// TIA Portal V19 export
DATA_BLOCK "A0201_Profilatrice_RegolazioneFormato_PERS"   // DB70
// stored: MemoryReserve 100
   VAR RETAIN
      Par_Machine { ExternalAccessible := 'False'; ExternalVisible := 'False'; ExternalWritable := 'False'} : Struct
         Passaggio02_MaxDisallineamentoAXs : Real := 0.5;   // (Controllo disabilitato se <= 0)
         Passaggio14_MaxDisallineamentoAXs : Real := 0.5;   // (Controllo disabilitato se <= 0)
         Passaggio17_MaxDisallineamentoAXs : Real := 0.5;   // (Controllo disabilitato se <= 0)
         Passaggio18_MaxDisallineamentoAXs : Real := 0.5;   // (Controllo disabilitato se <= 0)
         AxD_AutoSpeed : Real := 100.0;
      END_STRUCT;
      Par_Enc : Array[1..14] of "PosFbk_RTN";
      Par_D { S7_SetPoint := 'True'} : Array[1..6] of "Positioning_DOL_Machine_Par";
      Par_M { S7_SetPoint := 'True'} : Array[7..14] of "Positioning_MOL_Machine_Par";
      Pers_D { S7_SetPoint := 'True'} : Array[1..6] of "Positioning_DOL_Machine_Pers_Data";
      Pers_M { S7_SetPoint := 'True'} : Array[7..14] of "Positioning_MOL_Machine_Pers_Data";
   END_VAR
BEGIN
   Par_Enc[1].Preset.Pulses := 1_563_135_560;
   Par_Enc[2].Preset.Pulses := 283_648_312;
   Par_Enc[3].Preset.Pulses := -86_148_656;
   Par_Enc[4].Preset.Pulses := -1_788_471_592;
   Par_Enc[5].Preset.Pulses := -125_649_756;
   Par_Enc[6].Preset.Pulses := -399_566_752;
   Par_Enc[7].Preset.Pulses := 1_163_925_416;
   Par_Enc[8].Preset.Pulses := -87_886_012;
   Par_Enc[9..10].Preset.Pulses := 0;
   Par_Enc[11].Preset.Pulses := -1_797_037_560;
   Par_Enc[12].Preset.Pulses := 791_619_740;
   Par_Enc[13].Preset.Pulses := -29_607_776;
   Par_Enc[14].Preset.Pulses := 834_749_188;
   Par_Enc[1].Preset.Units := 91.6499938964844;
   Par_Enc[2].Preset.Units := 106.899987792969;
   Par_Enc[3].Preset.Units := 152.159987792969;
   Par_Enc[4].Preset.Units := 59.5800061035156;
   Par_Enc[5].Preset.Units := 144.899987792969;
   Par_Enc[6].Preset.Units := 60.4;
   Par_Enc[7].Preset.Units := 1.40000305175781;
   Par_Enc[8].Preset.Units := 0.700003051757818;
   Par_Enc[9..10].Preset.Units := 0.0;
   Par_Enc[11..12].Preset.Units := 1.5000015258789;
   Par_Enc[13..14].Preset.Units := 1.50000305175782;
   Par_Enc[1..6].Config.Resolution := 0.2;
   Par_Enc[7..14].Config.Resolution := -1.0;
   Par_D[1..6].PosTolerance := 0.05;
   Par_D[1..2].Minus_Limit := 70.0;
   Par_D[3..6].Minus_Limit := 30.0;
   Par_D[1].Plus_Limit := 162.0;
   Par_D[2].Plus_Limit := 161.0;
   Par_D[3..6].Plus_Limit := 156.5;
   Par_D[1..6].PreCutOff := 0.1;
   Par_D[1..6].PreEndLowSpeed := 2.0;
   Par_D[1..6].PreEndMedSpeed := 5.0;
   Par_D[1..6].LowSpeed := 20.0;
   Par_D[1..6].MedSpeed := 60.0;
   Par_D[1..6].HighSpeed := 60.0;
   Par_D[1..6].Man_Speed := 100.0;
   Par_M[7..14].PosTolerance := 0.05;
   Par_M[7..14].DelayInPosition := T#100MS;
   Par_M[7..14].Minus_Limit := 0.0;
   Par_M[7..14].Plus_Limit := 5.1;
   Par_M[7..14].PreCutOff := 0.03;
   Pers_D[1..6].AxisHomed := TRUE;
   Pers_M[7..14].AxisHomed := TRUE;
END_DATA_BLOCK
